PROGRAM Initial_POU
VAR
	nStep	:INT;
	strText	:STRING;
	aryBit	:ARRAY [0..100] OF BOOL;
	dwError: DWORD;
	tmrDelay,tmrDone	:TON;
END_VAR

CASE nStep OF
	0:
		tmrDelay(IN:=FALSE);
		tmrDone(IN:=FALSE);
		strText:= 'Intiail Runing';
		EventLogger.eEventType		:= 2;
		EventLogger.strEventText	:= 'Ini. Execute! ';	
		EventLogger();
		OP.xInitialDone				:=FALSE;
		nStep:= 5;
		IF LEN(RunParameter.strName) = 0 THEN
			nStep			:= 90;
			EventLogger.eEventType		:= 3;
			EventLogger.strEventText	:= 'Recipe Not Find ';	
			EventLogger();
			strText			:= 'Ini.Recipe Not Find';
		END_IF;
	5:
		tmrDelay(IN:=TRUE,PT:=T#5S);		
		IF tmrDelay.Q THEN
			strText:= 'Ini.Recipe Time Up ';
			EventLogger.eEventType		:= 3;
			EventLogger.strEventText	:= 'Recipe TimeUp ';	
			EventLogger();
			tmrDelay(IN:=FALSE);
			nStep			:= 90;
		END_IF	
			dwError:= RecipeManCommands.LoadAndWriteRecipe(RecipeDefinitionName:='Recipes' , RecipeName:=RunParameter.strName);	
			IF dwError = 0 THEN
				RunParameter	:= Edit_Parameter;
				strText:= 'Ini.Run Home ';
				nStep			:= 6;
				ELSE
				nStep			:= 90;
				strText:= 'Ini.Recipe Not Find';
				EventLogger.eEventType		:= 3;
				EventLogger.strEventText	:= 'Recipe Not Find ';	
				EventLogger();
			END_IF
	6:
		MainControl.ErrorReset();
		IF Air_Signal THEN
			nStep			:= 10;
			ELSE
			nStep			:= 90;
			strText:= 'Ini. Insuff. Air Pressure ';
			EventLogger.eEventType		:= 3;
			EventLogger.strEventText	:= ' Insuff. Air Pressure  ';	
			EventLogger();
		END_IF;		
	10:
		tmrDelay(IN:=TRUE,PT:=T#50S);		
		IF tmrDelay.Q THEN
			strText:= 'RB Init.TimeUp ';
			EventLogger.eEventType		:= 3;
			EventLogger.strEventText	:= ' RB Init.TimeUp ';	
			EventLogger();
			tmrDelay(IN:=FALSE);
			nStep			:= 90;
		END_IF	
	
		
		tmrDone(IN:= aryBit[7] AND aryBit[8],PT:=T#0.1S );
		aryBit[7]:=RB_CS.Initialization();
		aryBit[8]:=RB_KR.Initialization();					
		IF 	RB_CS.CommandError THEN
			strText:= 'RB Init. CS BOX Error ';
			EventLogger.eEventType		:= 3;
			EventLogger.strEventText	:= 'RB Init. CS BOX Error';	
			EventLogger();
			tmrDelay(IN:=FALSE);
			nStep			:= 90;
		END_IF
		IF tmrDone.Q THEN
			tmrDelay(IN:=FALSE);
			nStep	:= 20;	
		END_IF
	20:
		aryBit[0]:=M_DualServo.Initialization(FALSE);
		aryBit[1]:=M_Openbox1.Initialization(FALSE);
		aryBit[2]:=M_Sealing2.Initialization(FALSE);
		aryBit[3]:=M_LoadPic3.Initialization(FALSE);
		aryBit[4]:=M_UnloadNG4.Initialization(FALSE);
		aryBit[5]:=M_StackComv5.Initialization(FALSE);
		aryBit[6]:=M_RBStack6.Initialization(FALSE);
		tmrDelay(IN:=TRUE,PT:=T#50S);		
		IF tmrDelay.Q THEN
			strText:= 'Init. TimeUp ';
			EventLogger.eEventType		:= 3;
			EventLogger.strEventText	:= 'Hardware TimeUp';	
			EventLogger();
			tmrDelay(IN:=FALSE);
			nStep			:= 99;	
		END_IF
		tmrDone(IN:= aryBit[0] AND aryBit[1] AND aryBit[2] AND aryBit[3] AND aryBit[4] AND aryBit[5] AND aryBit[6] ,PT:=T#0.1S);
		IF  tmrDone.q THEN
			tmrDone(IN:=FALSE);
			tmrDelay(IN:=FALSE);
			EventLogger.eEventType		:= 1;
			EventLogger.strEventText	:= 'Intil. Complete';	
			EventLogger();
			strText:= 'Int.Finished';
			nStep			:= 50;
		END_IF;
		
	50:
		OP.xInitialDone	:= TRUE;	
	90:		
		EventLogger.eEventType		:= 3;
		EventLogger.strEventText	:= 'Ini. Cancel!';	
		EventLogger();	
		nStep			:= 91;	
END_CASE

METHOD FB_init : BOOL
VAR_INPUT
	bInitRetains : BOOL; // if TRUE, the retain variables are initialized (warm start / cold start)
	bInCopyCode : BOOL;  // if TRUE, the instance afterwards gets moved into the copy code (online change)
END_VAR
nStep	:= 0;
strText	:= '';
END_METHOD

END_PROGRAM

(* stored: Version 1.1.0.1, ProductVersion 3.1.4024.16
   POU Initial_POU: Id {9593bfb5-296d-4592-9257-2c0aff8b49cd}, SpecialFunc None
   Method FB_init: Id {f0e1d5c9-cb6f-4d69-9756-baed2e282f23} *)
